PROGRAM PRG_CohapTest
VAR
END_VAR

ACTION A_InitCohapMethodParams:
strDeviceName := 'Device12133';

readSerialNumber_inpuparams[0].strKey := 'channel';
readSerialNumber_inpuparams[0].strValue := '1';
readSerialNumber_inpuparams[1].strKey := '';
readSerialNumber_inpuparams[1].strValue := '';
readSerialNumber_inpuparams[2].strKey := '';
readSerialNumber_inpuparams[2].strValue := '';

readSerialNumber_expoutparamlist[0].enumDataType := E_DataType.DT_ULINT;
readSerialNumber_expoutparamlist[0].strVarName := 'serialnumber';
readSerialNumber_expoutparamlist[1].enumDataType := E_DataType.DT_STRING;
readSerialNumber_expoutparamlist[1].strVarName := 'stringserialno';
readSerialNumber_expoutparamlist[2].enumDataType := E_DataType.DT_STRING;
readSerialNumber_expoutparamlist[2].strVarName := '';


ReadDeviceOutput_inpuparams[0].strKey := 'channel';
ReadDeviceOutput_inpuparams[0].strValue := '1';
ReadDeviceOutput_inpuparams[1].strKey := '';
ReadDeviceOutput_inpuparams[1].strValue := '';
ReadDeviceOutput_inpuparams[2].strKey := '';
ReadDeviceOutput_inpuparams[2].strValue := '';

ReadDeviceOutput_expoutparamlist[0].enumDataType := E_DataType.DT_INT;
ReadDeviceOutput_expoutparamlist[0].strVarName := 'P1data';
ReadDeviceOutput_expoutparamlist[1].enumDataType := E_DataType.DT_INT;
ReadDeviceOutput_expoutparamlist[1].strVarName := 'P1out';
ReadDeviceOutput_expoutparamlist[2].enumDataType := E_DataType.DT_INT;
ReadDeviceOutput_expoutparamlist[2].strVarName := 'P2data';
ReadDeviceOutput_expoutparamlist[3].enumDataType := E_DataType.DT_INT;
ReadDeviceOutput_expoutparamlist[3].strVarName := 'P2out';
ReadDeviceOutput_expoutparamlist[4].enumDataType := E_DataType.DT_INT;
ReadDeviceOutput_expoutparamlist[4].strVarName := 'T1data';
ReadDeviceOutput_expoutparamlist[5].enumDataType := E_DataType.DT_INT;
ReadDeviceOutput_expoutparamlist[5].strVarName := 'T1out';
ReadDeviceOutput_expoutparamlist[6].enumDataType := E_DataType.DT_INT;
ReadDeviceOutput_expoutparamlist[6].strVarName := 'T2data';
ReadDeviceOutput_expoutparamlist[7].enumDataType := E_DataType.DT_INT;
ReadDeviceOutput_expoutparamlist[7].strVarName := 'T2out';

PowerUp_inpuparams[0].strKey := 'channel';
PowerUp_inpuparams[0].strValue := '1';
PowerUp_inpuparams[1].strKey := 'supplyVoltage';
PowerUp_inpuparams[1].strValue := '5.0';
PowerUp_inpuparams[2].strKey := '';
PowerUp_inpuparams[2].strValue := '';

PowerUp_expoutparamlist[0].enumDataType := E_DataType.DT_DOUBLE;
PowerUp_expoutparamlist[0].strVarName := 'Vsupply';
PowerUp_expoutparamlist[1].enumDataType := E_DataType.DT_DOUBLE;
PowerUp_expoutparamlist[1].strVarName := 'current';
PowerUp_expoutparamlist[2].enumDataType := E_DataType.DT_STRING;
PowerUp_expoutparamlist[2].strVarName := '';

PowerDown_inpuparams[0].strKey := 'channel';
PowerDown_inpuparams[0].strValue := '1';
PowerDown_inpuparams[1].strKey := '';
PowerDown_inpuparams[1].strValue := '';
PowerDown_inpuparams[2].strKey := '';
PowerDown_inpuparams[2].strValue := '';

PowerDown_expoutparamlist[0].enumDataType := E_DataType.DT_STRING;
PowerDown_expoutparamlist[0].strVarName := '';
PowerDown_expoutparamlist[1].enumDataType := E_DataType.DT_STRING;
PowerDown_expoutparamlist[1].strVarName := '';
PowerDown_expoutparamlist[2].enumDataType := E_DataType.DT_STRING;
PowerDown_expoutparamlist[2].strVarName := '';

TestDummy_inpuparams[0].strKey := 'channel';
TestDummy_inpuparams[0].strValue := '1';
TestDummy_inpuparams[1].strKey := 'bInput';
TestDummy_inpuparams[1].strValue := 'FALSE';
TestDummy_inpuparams[2].strKey := '';
TestDummy_inpuparams[2].strValue := '';

TestDummy_expoutparamlist[0].enumDataType := E_DataType.DT_STRING;
TestDummy_expoutparamlist[0].strVarName := 'serialno';
TestDummy_expoutparamlist[1].enumDataType := E_DataType.DT_DOUBLE;
TestDummy_expoutparamlist[1].strVarName := 'Voltage';
TestDummy_expoutparamlist[2].enumDataType := E_DataType.DT_BOOL;
TestDummy_expoutparamlist[2].strVarName := 'MethodResponse';
TestDummy_expoutparamlist[3].enumDataType := E_DataType.DT_UINT;
TestDummy_expoutparamlist[3].strVarName := 'current';
TestDummy_expoutparamlist[4].enumDataType := E_DataType.DT_STRING;
TestDummy_expoutparamlist[4].strVarName := 'P1status';
TestDummy_expoutparamlist[5].enumDataType := E_DataType.DT_STRING;
TestDummy_expoutparamlist[5].strVarName := 'P2status';

TestDummy2_inpuparams[0].strKey := 'channel';
TestDummy2_inpuparams[0].strValue := '1';
TestDummy2_inpuparams[1].strKey := 'Input2';
TestDummy2_inpuparams[1].strValue := 'dummyimput2';
TestDummy2_inpuparams[2].strKey := '';
TestDummy2_inpuparams[2].strValue := '';

TestDummy2_expoutparamlist[0].enumDataType := E_DataType.DT_INT;
TestDummy2_expoutparamlist[0].strVarName := 'output1';
TestDummy2_expoutparamlist[1].enumDataType := E_DataType.DT_STRING;
TestDummy2_expoutparamlist[1].strVarName := 'output2';
TestDummy2_expoutparamlist[2].enumDataType := E_DataType.DT_ULINT;
TestDummy2_expoutparamlist[2].strVarName := 'fastchannel1';
TestDummy2_expoutparamlist[3].enumDataType := E_DataType.DT_ULINT;
TestDummy2_expoutparamlist[3].strVarName := 'fastchannel2';
TestDummy2_expoutparamlist[4].enumDataType := E_DataType.DT_STRING;
TestDummy2_expoutparamlist[4].strVarName := 'fastchannel3';
TestDummy2_expoutparamlist[5].enumDataType := E_DataType.DT_INT;
TestDummy2_expoutparamlist[5].strVarName := 'fastchannel4';
TestDummy2_expoutparamlist[6].enumDataType := E_DataType.DT_ULINT;
TestDummy2_expoutparamlist[6].strVarName := 'fastchannel5';
TestDummy2_expoutparamlist[7].enumDataType := E_DataType.DT_ULINT;
TestDummy2_expoutparamlist[7].strVarName := 'fastchannel6';
TestDummy2_expoutparamlist[8].enumDataType := E_DataType.DT_STRING;
TestDummy2_expoutparamlist[8].strVarName := 'fastchannel7';
TestDummy2_expoutparamlist[9].enumDataType := E_DataType.DT_INT;
TestDummy2_expoutparamlist[9].strVarName := 'fastchannel8';

//TestDummy2_outputparams[0].strKey := '';
//TestDummy2_outputparams[0].strValue := '';
//TestDummy2_outputparams[1].strKey := '';
//TestDummy2_outputparams[1].strValue := '';
//TestDummy2_outputparams[2].strKey := '';
//TestDummy2_outputparams[2].strValue := '';
//TestDummy2_outputparams[3].strKey := '';
//TestDummy2_outputparams[3].strValue := '';
//TestDummy2_outputparams[4].strKey := '';
//TestDummy2_outputparams[4].strValue := '';
//TestDummy2_outputparams[5].strKey := '';
//TestDummy2_outputparams[5].strValue := '';
//TestDummy2_outputparams[6].strKey := '';
//TestDummy2_outputparams[6].strValue := '';
//TestDummy2_outputparams[7].strKey := '';
//TestDummy2_outputparams[7].strValue := '';
//TestDummy2_outputparams[8].strKey := '';
//TestDummy2_outputparams[8].strValue := '';
//TestDummy2_outputparams[9].strKey := '';
//TestDummy2_outputparams[9].strValue := '';

init_inpuparams[0].strKey := 'VSupply';
init_inpuparams[0].strValue := '5.0';
init_inpuparams[1].strKey := '';
init_inpuparams[1].strValue := '';
init_inpuparams[2].strKey := '';
init_inpuparams[2].strValue := '';

init_expoutparamlist[0].enumDataType := E_DataType.DT_STRING;
init_expoutparamlist[0].strVarName := 'returnMsg';
init_expoutparamlist[1].enumDataType := E_DataType.DT_STRING;
init_expoutparamlist[1].strVarName := '';
init_expoutparamlist[2].enumDataType := E_DataType.DT_STRING;
init_expoutparamlist[2].strVarName := '';

getSICAndChannelCardVersions_inpuparams[0].strKey := 'channel';
getSICAndChannelCardVersions_inpuparams[0].strValue := '1';
getSICAndChannelCardVersions_inpuparams[1].strKey := '';
getSICAndChannelCardVersions_inpuparams[1].strValue := '';
getSICAndChannelCardVersions_inpuparams[2].strKey := '';
getSICAndChannelCardVersions_inpuparams[2].strValue := '';

getSICAndChannelCardVersions_expoutparamlist[0].enumDataType := E_DataType.DT_STRING;
getSICAndChannelCardVersions_expoutparamlist[0].strVarName := 'SICVersion';
getSICAndChannelCardVersions_expoutparamlist[1].enumDataType := E_DataType.DT_STRING;
getSICAndChannelCardVersions_expoutparamlist[1].strVarName := 'COHAPChannelCardVersion';
getSICAndChannelCardVersions_expoutparamlist[2].enumDataType := E_DataType.DT_STRING;
getSICAndChannelCardVersions_expoutparamlist[2].strVarName := '';

getDLLVersions_inpuparams[0].strKey := '';
getDLLVersions_inpuparams[0].strValue := '';
getDLLVersions_inpuparams[1].strKey := '';
getDLLVersions_inpuparams[1].strValue := '';
getDLLVersions_inpuparams[2].strKey := '';
getDLLVersions_inpuparams[2].strValue := '';

getDLLVersions_expoutparamlist[0].enumDataType := E_DataType.DT_STRING;
getDLLVersions_expoutparamlist[0].strVarName := 'DUT12133DLLVersion';
getDLLVersions_expoutparamlist[1].enumDataType := E_DataType.DT_STRING;
getDLLVersions_expoutparamlist[1].strVarName := 'MUPeT12133DLLVersion';
getDLLVersions_expoutparamlist[2].enumDataType := E_DataType.DT_STRING;
getDLLVersions_expoutparamlist[2].strVarName := 'HALDLLVersion';


initDUT_inpuparams[0].strKey := 'channel';
initDUT_inpuparams[0].strValue := '1';
initDUT_inpuparams[1].strKey := 'supplyVoltage';
initDUT_inpuparams[1].strValue := '5.0';
initDUT_inpuparams[2].strKey := '';
initDUT_inpuparams[2].strValue := '';

initDUT_expoutparamlist[0].enumDataType := E_DataType.DT_STRING;
initDUT_expoutparamlist[0].strVarName := '';
initDUT_expoutparamlist[1].enumDataType := E_DataType.DT_STRING;
initDUT_expoutparamlist[1].strVarName := '';
initDUT_expoutparamlist[2].enumDataType := E_DataType.DT_STRING;
initDUT_expoutparamlist[2].strVarName := '';


readFastChannelData_inputparams[0].strKey := 'channel';
readFastChannelData_inputparams[0].strValue := '1';
readFastChannelData_inputparams[1].strKey := '';
readFastChannelData_inputparams[1].strValue := '';
readFastChannelData_inputparams[2].strKey := '';
readFastChannelData_inputparams[2].strValue := '';

readFastChannelData_expoutparamlist[0].enumDataType := E_DataType.DT_UINT;
readFastChannelData_expoutparamlist[0].strVarName := 'FastChannel1Data';
readFastChannelData_expoutparamlist[1].enumDataType := E_DataType.DT_UINT;
readFastChannelData_expoutparamlist[1].strVarName := 'FastChannel2Data';
readFastChannelData_expoutparamlist[2].enumDataType := E_DataType.DT_STRING;
readFastChannelData_expoutparamlist[2].strVarName := 'FastChannel1Status';
readFastChannelData_expoutparamlist[3].enumDataType := E_DataType.DT_STRING;
readFastChannelData_expoutparamlist[3].strVarName := 'FastChannel2Status';


InitLot_inputparams[0].strKey := 'deviceID';
InitLot_inputparams[0].strValue := '52EMB01-01';
InitLot_inputparams[1].strKey := 'lotID';
InitLot_inputparams[1].strValue := '123';
InitLot_inputparams[2].strKey := 'equipmentID';
InitLot_inputparams[2].strValue := '1';
InitLot_inputparams[3].strKey := 'testKind';
InitLot_inputparams[3].strValue := '1';

t1Precal_inputparams[0].strKey := 'channel';
t1Precal_inputparams[0].strValue := '1';
t1Precal_inputparams[1].strKey := 'deviceID';
t1Precal_inputparams[1].strValue := '52EMB01-01';
t1Precal_inputparams[2].strKey := 'temperature';
t1Precal_inputparams[2].strValue := '-25';
t1Precal_inputparams[3].strKey := 'force';
t1Precal_inputparams[3].strValue := '0';
 
t1Step2_inputparams[0].strKey := 'deviceID';
t1Step2_inputparams[0].strValue := '52EMB01-01';
t1Step2_inputparams[1].strKey := 'temperature';
t1Step2_inputparams[1].strValue := '-25';
t1Step2_inputparams[2].strKey := 'force';
t1Step2_inputparams[2].strValue := '40';
 
t1Step3_inputparams[0].strKey := 'deviceID';
t1Step3_inputparams[0].strValue := '52EMB01-01';
t1Step3_inputparams[2].strKey := 'temperature';
t1Step3_inputparams[2].strValue := '-25';
t1Step3_inputparams[3].strKey := 'force';
t1Step3_inputparams[3].strValue := '0';
END_ACTION

METHOD M_TestCohapLibrary : BOOL
VAR_INPUT
END_VAR
VAR
	//Testing Cohap Related Vars

	//Initialize Only	
	MyCohapTest : FB_COHAP;
	bInitializeCohapSystem: BOOL;
	bRes_CohapConnected: BOOL;

	//Execute RunImpMethods Only	;
	bExecuteRunImpMethods: BOOL;
	bRes_RunImpMethods: BOOL;

	//Set Current Device Instance
	bSetCurrentDevice_Cohap : BOOL;
	bRes_SetCurrentDevice : BOOL;
	//Input Params
	strDeviceName : STRING;
	
	//RunCommand
	bRunCommandCohapSystem : BOOL;
	bRes_RunCommand : BOOL;
	//Input Params
	strMethodName : STRING;
	RunCom_InpuParams : T_CohapParameterList;
	RunCom_ExpOutParamList : ARRAY[0..9] OF ST_ReturnParamsInfo;
	//Output Params
	RunCom_OutputParams : T_CohapParameterList;
	
	//DummyTest Dictionary Prep for RunCommand Execution
	RC_DT_InpPar : T_CohapParameterList;
	RC_DT_ExpOutPL : ARRAY[0..9] OF ST_ReturnParamsInfo;
	
	CohapMethodStrings : TMethodNames_Cohap;
	CohapMethodControls : TMethod_Controls;
//	fbCohapHandler1: FB_COHAP;

///////////////////////////////

	// For readSerialNumber
	readSerialNumber_inpuparams : T_CohapParameterList;
	readSerialNumber_expoutparamlist : ARRAY[0..9] OF ST_ReturnParamsInfo;
	readSerialNumber_outputparams : T_CohapParameterList;
	
	// For ReadDeviceOutput
	ReadDeviceOutput_inpuparams : T_CohapParameterList;
	ReadDeviceOutput_expoutparamlist : ARRAY[0..9] OF ST_ReturnParamsInfo;
	ReadDeviceOutput_outputparams : T_CohapParameterList;

	
	// For PowerUp
	PowerUp_inpuparams : T_CohapParameterList;
	PowerUp_expoutparamlist : ARRAY[0..9] OF ST_ReturnParamsInfo;
	PowerUp_outputparams : T_CohapParameterList;
	
	// For PowerDown
	PowerDown_inpuparams : T_CohapParameterList;
	PowerDown_expoutparamlist : ARRAY[0..9] OF ST_ReturnParamsInfo;
	PowerDown_outputparams : T_CohapParameterList;
	
	// For TestDummy
	TestDummy_inpuparams : T_CohapParameterList;
	TestDummy_expoutparamlist : ARRAY[0..9] OF ST_ReturnParamsInfo;
	TestDummy_outputparams : T_CohapParameterList;
	
	// For TestDummy2
	TestDummy2_inpuparams : T_CohapParameterList;
	TestDummy2_expoutparamlist : ARRAY[0..9] OF ST_ReturnParamsInfo;
	TestDummy2_outputparams : T_CohapParameterList;
	
	// For init
	init_inpuparams : T_CohapParameterList;
	init_expoutparamlist : ARRAY[0..9] OF ST_ReturnParamsInfo;
	init_outputparams : T_CohapParameterList;
	
	// For getSICAndChannelCardVersions
	getSICAndChannelCardVersions_inpuparams : T_CohapParameterList;
	getSICAndChannelCardVersions_expoutparamlist : ARRAY[0..9] OF ST_ReturnParamsInfo;
	getSICAndChannelCardVersions_outputparams : T_CohapParameterList;
	
	// For getDLLVersions
	getDLLVersions_inpuparams : T_CohapParameterList;
	getDLLVersions_expoutparamlist : ARRAY[0..9] OF ST_ReturnParamsInfo;
	getDLLVersions_outputparams : T_CohapParameterList;
	
	// For initDUT
	initDUT_inpuparams : T_CohapParameterList;
	initDUT_expoutparamlist : ARRAY[0..9] OF ST_ReturnParamsInfo;
	initDUT_outputparams : T_CohapParameterList;
	
	//For Fast Channel Data
	readFastChannelData_inputparams : T_CohapParameterList;
	readFastChannelData_expoutparamlist : ARRAY[0..9] OF ST_ReturnParamsInfo;
	readFastChannelData_outputparams : T_CohapParameterList;

	// For T1 Step 1 Calibration
	t1Step1_inpuparams : T_CohapParameterList;
	t1Step1_expoutparamlist : ARRAY[0..9] OF ST_ReturnParamsInfo;
	t1Step1_outputparams : T_CohapParameterList;
	
//	// For T1 Step 2 Calibration
//	t1Step2_inpuparams : T_CohapParameterList;
//	t1Step2_expoutparamlist : ARRAY[0..9] OF ST_ReturnParamsInfo;
//	t1Step2_outputparams : T_CohapParameterList;
	
//	// For T1 Step 3 Calibration
//	t1Step3_inpuparams : T_CohapParameterList;
//	t1Step3_expoutparamlist : ARRAY[0..9] OF ST_ReturnParamsInfo;
//	t1Step3_outputparams : T_CohapParameterList;
	
	// For T2 Step 1 Calibration
	t2Step1_inpuparams : T_CohapParameterList;
	t2Step1_expoutparamlist : ARRAY[0..9] OF ST_ReturnParamsInfo;
	t2Step1_outputparams : T_CohapParameterList;
	
	// For T2 Step 2 Calibration
	t2Step2_inpuparams : T_CohapParameterList;
	t2Step2_expoutparamlist : ARRAY[0..9] OF ST_ReturnParamsInfo;
	t2Step2_outputparams : T_CohapParameterList;
	
	// For T2 Step 3 Calibration
	t2Step3_inpuparams : T_CohapParameterList;
	t2Step3_expoutparamlist : ARRAY[0..9] OF ST_ReturnParamsInfo;
	t2Step3_outputparams : T_CohapParameterList;
	
	// InitLot Device12133 class in Mech Device Lib Calibration
	InitLot_inputparams : T_CohapParameterList;
	InitLot_expoutparamlist : ARRAY[0..9] OF ST_ReturnParamsInfo;
	InitLot_outputparams : T_CohapParameterList;
	
//	//For Init Lot
//	InitLot_inputparams : T_CohapParameterList;
//	InitLot_expoutparamlist : ARRAY[0..9] OF ST_ReturnParamsInfo;
//	InitLot_outputparams : T_CohapParameterList;	
	// For T1 Step 1 Calibration
	t1Precal_inputparams : T_CohapParameterList;
	t1Precal_expoutparamlist : ARRAY[0..9] OF ST_ReturnParamsInfo;
	t1Precal_outputparams : T_CohapParameterList;
	// For T1 Step 2 Calibration
	t1Step2_inputparams : T_CohapParameterList;
	t1Step2_expoutparamlist : ARRAY[0..9] OF ST_ReturnParamsInfo;
	t1Step2_outputparams : T_CohapParameterList;
	// For T1 Step 3 Calibration
	t1Step3_inputparams : T_CohapParameterList;
	t1Step3_expoutparamlist : ARRAY[0..9] OF ST_ReturnParamsInfo;
	t1Step3_outputparams : T_CohapParameterList;
END_VAR
VAR_INST // added by the converter: edge detectors and wires of the graphical bodies
    _w1, _w2, _w3, _w4, _w5, _w6, _w7, _w8, _w9, _w10, _w11, _w12, _w13, _w14, _w15, _w16, _w17, _w18, _w19, _w20, _w21, _w22, _w23, _w24, _w25, _w26, _w27, _w28, _w29, _w30, _w31, _w32, _w33, _w34, _w35, _w36, _w37, _w38, _w39, _w40 : BOOL;
END_VAR
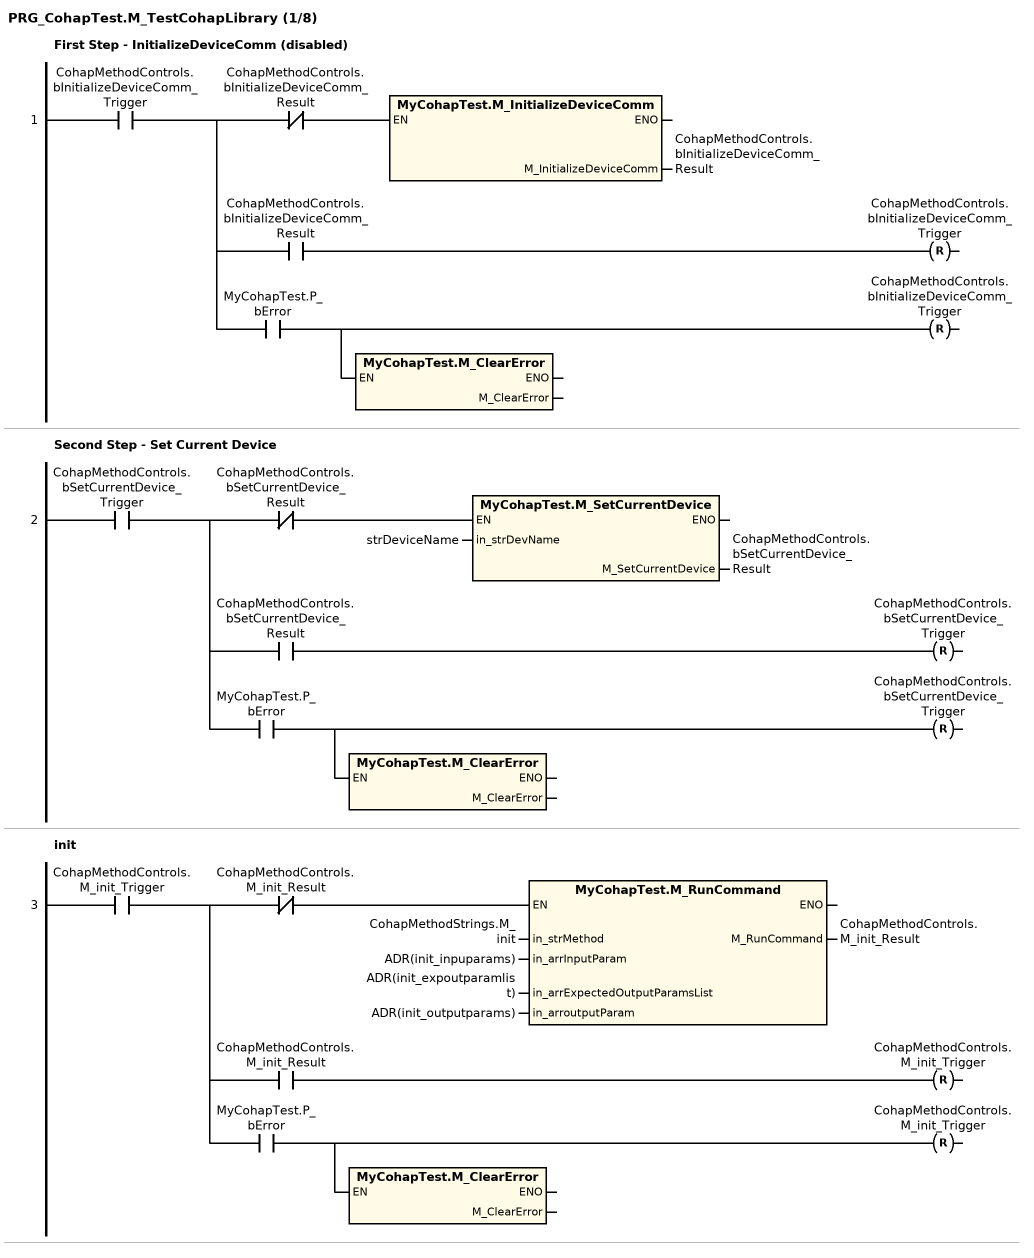
// NETWORK 1: First Step - InitializeDeviceComm (disabled)
// _w1 := CohapMethodControls.bInitializeDeviceComm_Trigger;
// IF _w1 AND NOT CohapMethodControls.bInitializeDeviceComm_Result THEN
//     CohapMethodControls.bInitializeDeviceComm_Result := MyCohapTest.M_InitializeDeviceComm();
// END_IF
// CohapMethodControls.bInitializeDeviceComm_Trigger R= _w1 AND CohapMethodControls.bInitializeDeviceComm_Result;
// _w2 := _w1 AND MyCohapTest.P_bError;
// CohapMethodControls.bInitializeDeviceComm_Trigger R= _w2;
// IF _w2 THEN MyCohapTest.M_ClearError(); END_IF

// NETWORK 2: Second Step - Set Current Device
_w3 := CohapMethodControls.bSetCurrentDevice_Trigger;
IF _w3 AND NOT CohapMethodControls.bSetCurrentDevice_Result THEN
    CohapMethodControls.bSetCurrentDevice_Result := MyCohapTest.M_SetCurrentDevice(in_strDevName := strDeviceName);
END_IF
CohapMethodControls.bSetCurrentDevice_Trigger R= _w3 AND CohapMethodControls.bSetCurrentDevice_Result;
_w4 := _w3 AND MyCohapTest.P_bError;
CohapMethodControls.bSetCurrentDevice_Trigger R= _w4;
IF _w4 THEN MyCohapTest.M_ClearError(); END_IF

// NETWORK 3: init
_w5 := CohapMethodControls.M_init_Trigger;
IF _w5 AND NOT CohapMethodControls.M_init_Result THEN
    CohapMethodControls.M_init_Result := MyCohapTest.M_RunCommand(in_strMethod := CohapMethodStrings.M_init, in_arrInputParam := ADR(init_inpuparams), in_arrExpectedOutputParamsList := ADR(init_expoutparamlist), in_arroutputParam := ADR(init_outputparams));
END_IF
CohapMethodControls.M_init_Trigger R= _w5 AND CohapMethodControls.M_init_Result;
_w6 := _w5 AND MyCohapTest.P_bError;
CohapMethodControls.M_init_Trigger R= _w6;
IF _w6 THEN MyCohapTest.M_ClearError(); END_IF

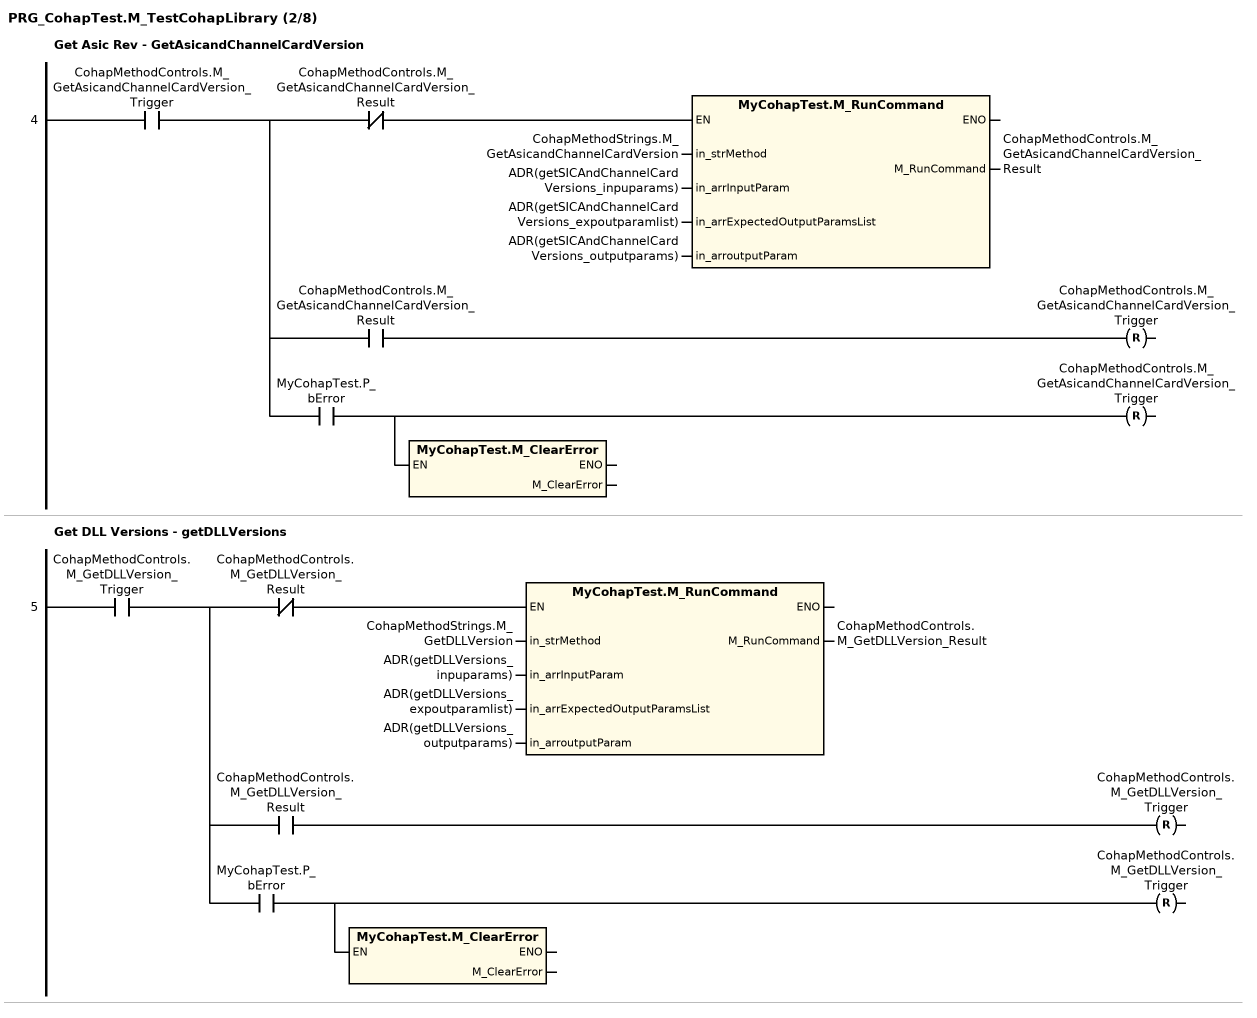
// NETWORK 4: Get Asic Rev - GetAsicandChannelCardVersion
_w7 := CohapMethodControls.M_GetAsicandChannelCardVersion_Trigger;
IF _w7 AND NOT CohapMethodControls.M_GetAsicandChannelCardVersion_Result THEN
    CohapMethodControls.M_GetAsicandChannelCardVersion_Result := MyCohapTest.M_RunCommand(in_strMethod := CohapMethodStrings.M_GetAsicandChannelCardVersion, in_arrInputParam := ADR(getSICAndChannelCardVersions_inpuparams), in_arrExpectedOutputParamsList := ADR(getSICAndChannelCardVersions_expoutparamlist), in_arroutputParam := ADR(getSICAndChannelCardVersions_outputparams));
END_IF
CohapMethodControls.M_GetAsicandChannelCardVersion_Trigger R= _w7 AND CohapMethodControls.M_GetAsicandChannelCardVersion_Result;
_w8 := _w7 AND MyCohapTest.P_bError;
CohapMethodControls.M_GetAsicandChannelCardVersion_Trigger R= _w8;
IF _w8 THEN MyCohapTest.M_ClearError(); END_IF

// NETWORK 5: Get DLL Versions - getDLLVersions
_w9 := CohapMethodControls.M_GetDLLVersion_Trigger;
IF _w9 AND NOT CohapMethodControls.M_GetDLLVersion_Result THEN
    CohapMethodControls.M_GetDLLVersion_Result := MyCohapTest.M_RunCommand(in_strMethod := CohapMethodStrings.M_GetDLLVersion, in_arrInputParam := ADR(getDLLVersions_inpuparams), in_arrExpectedOutputParamsList := ADR(getDLLVersions_expoutparamlist), in_arroutputParam := ADR(getDLLVersions_outputparams));
END_IF
CohapMethodControls.M_GetDLLVersion_Trigger R= _w9 AND CohapMethodControls.M_GetDLLVersion_Result;
_w10 := _w9 AND MyCohapTest.P_bError;
CohapMethodControls.M_GetDLLVersion_Trigger R= _w10;
IF _w10 THEN MyCohapTest.M_ClearError(); END_IF

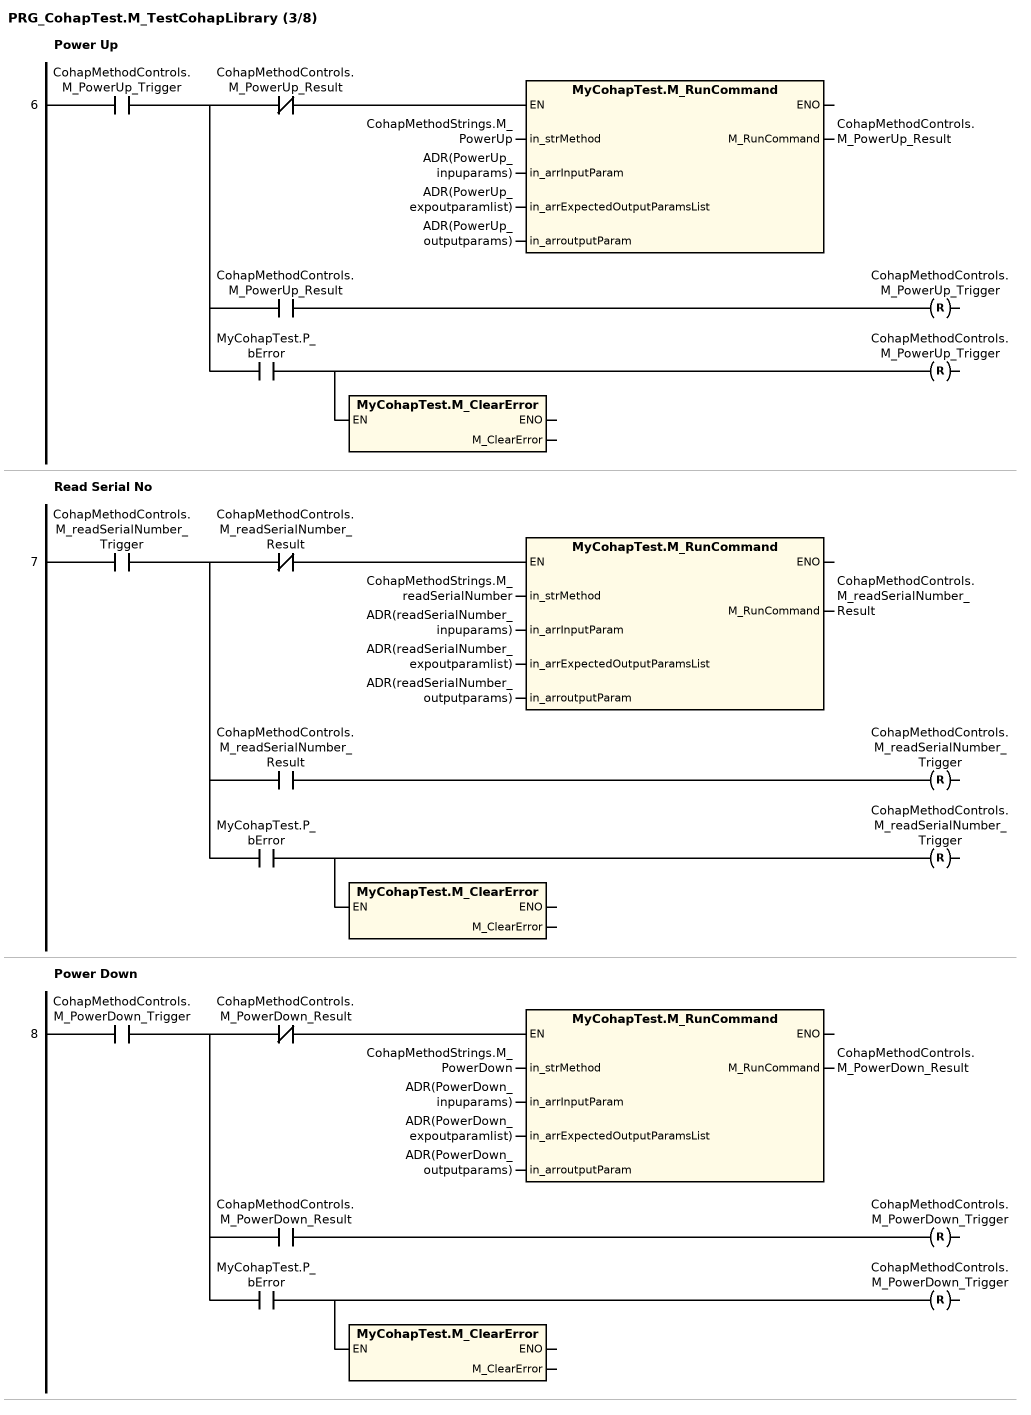
// NETWORK 6: Power Up
_w11 := CohapMethodControls.M_PowerUp_Trigger;
IF _w11 AND NOT CohapMethodControls.M_PowerUp_Result THEN
    CohapMethodControls.M_PowerUp_Result := MyCohapTest.M_RunCommand(in_strMethod := CohapMethodStrings.M_PowerUp, in_arrInputParam := ADR(PowerUp_inpuparams), in_arrExpectedOutputParamsList := ADR(PowerUp_expoutparamlist), in_arroutputParam := ADR(PowerUp_outputparams));
END_IF
CohapMethodControls.M_PowerUp_Trigger R= _w11 AND CohapMethodControls.M_PowerUp_Result;
_w12 := _w11 AND MyCohapTest.P_bError;
CohapMethodControls.M_PowerUp_Trigger R= _w12;
IF _w12 THEN MyCohapTest.M_ClearError(); END_IF

// NETWORK 7: Read Serial No
_w13 := CohapMethodControls.M_readSerialNumber_Trigger;
IF _w13 AND NOT CohapMethodControls.M_readSerialNumber_Result THEN
    CohapMethodControls.M_readSerialNumber_Result := MyCohapTest.M_RunCommand(in_strMethod := CohapMethodStrings.M_readSerialNumber, in_arrInputParam := ADR(readSerialNumber_inpuparams), in_arrExpectedOutputParamsList := ADR(readSerialNumber_expoutparamlist), in_arroutputParam := ADR(readSerialNumber_outputparams));
END_IF
CohapMethodControls.M_readSerialNumber_Trigger R= _w13 AND CohapMethodControls.M_readSerialNumber_Result;
_w14 := _w13 AND MyCohapTest.P_bError;
CohapMethodControls.M_readSerialNumber_Trigger R= _w14;
IF _w14 THEN MyCohapTest.M_ClearError(); END_IF

// NETWORK 8: Power Down
_w15 := CohapMethodControls.M_PowerDown_Trigger;
IF _w15 AND NOT CohapMethodControls.M_PowerDown_Result THEN
    CohapMethodControls.M_PowerDown_Result := MyCohapTest.M_RunCommand(in_strMethod := CohapMethodStrings.M_PowerDown, in_arrInputParam := ADR(PowerDown_inpuparams), in_arrExpectedOutputParamsList := ADR(PowerDown_expoutparamlist), in_arroutputParam := ADR(PowerDown_outputparams));
END_IF
CohapMethodControls.M_PowerDown_Trigger R= _w15 AND CohapMethodControls.M_PowerDown_Result;
_w16 := _w15 AND MyCohapTest.P_bError;
CohapMethodControls.M_PowerDown_Trigger R= _w16;
IF _w16 THEN MyCohapTest.M_ClearError(); END_IF

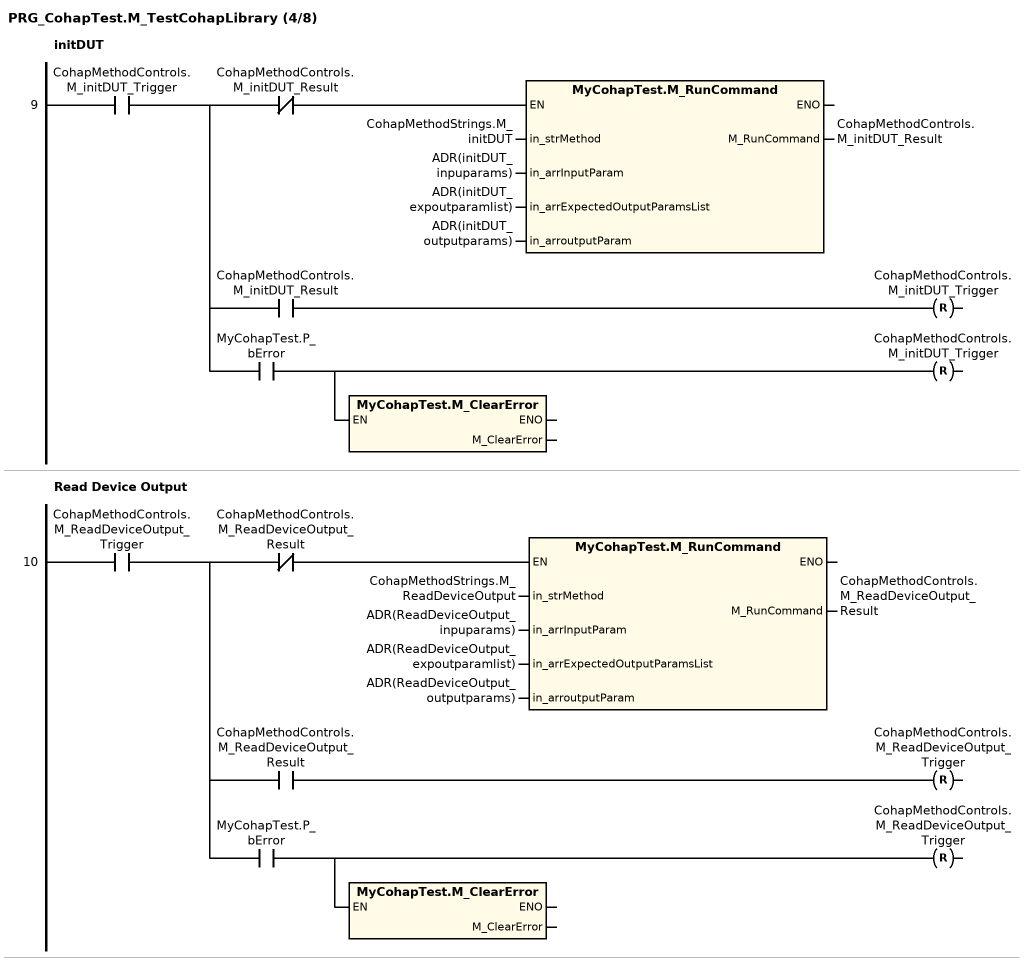
// NETWORK 9: initDUT
_w17 := CohapMethodControls.M_initDUT_Trigger;
IF _w17 AND NOT CohapMethodControls.M_initDUT_Result THEN
    CohapMethodControls.M_initDUT_Result := MyCohapTest.M_RunCommand(in_strMethod := CohapMethodStrings.M_initDUT, in_arrInputParam := ADR(initDUT_inpuparams), in_arrExpectedOutputParamsList := ADR(initDUT_expoutparamlist), in_arroutputParam := ADR(initDUT_outputparams));
END_IF
CohapMethodControls.M_initDUT_Trigger R= _w17 AND CohapMethodControls.M_initDUT_Result;
_w18 := _w17 AND MyCohapTest.P_bError;
CohapMethodControls.M_initDUT_Trigger R= _w18;
IF _w18 THEN MyCohapTest.M_ClearError(); END_IF

// NETWORK 10: Read Device Output
_w19 := CohapMethodControls.M_ReadDeviceOutput_Trigger;
IF _w19 AND NOT CohapMethodControls.M_ReadDeviceOutput_Result THEN
    CohapMethodControls.M_ReadDeviceOutput_Result := MyCohapTest.M_RunCommand(in_strMethod := CohapMethodStrings.M_ReadDeviceOutput, in_arrInputParam := ADR(ReadDeviceOutput_inpuparams), in_arrExpectedOutputParamsList := ADR(ReadDeviceOutput_expoutparamlist), in_arroutputParam := ADR(ReadDeviceOutput_outputparams));
END_IF
CohapMethodControls.M_ReadDeviceOutput_Trigger R= _w19 AND CohapMethodControls.M_ReadDeviceOutput_Result;
_w20 := _w19 AND MyCohapTest.P_bError;
CohapMethodControls.M_ReadDeviceOutput_Trigger R= _w20;
IF _w20 THEN MyCohapTest.M_ClearError(); END_IF

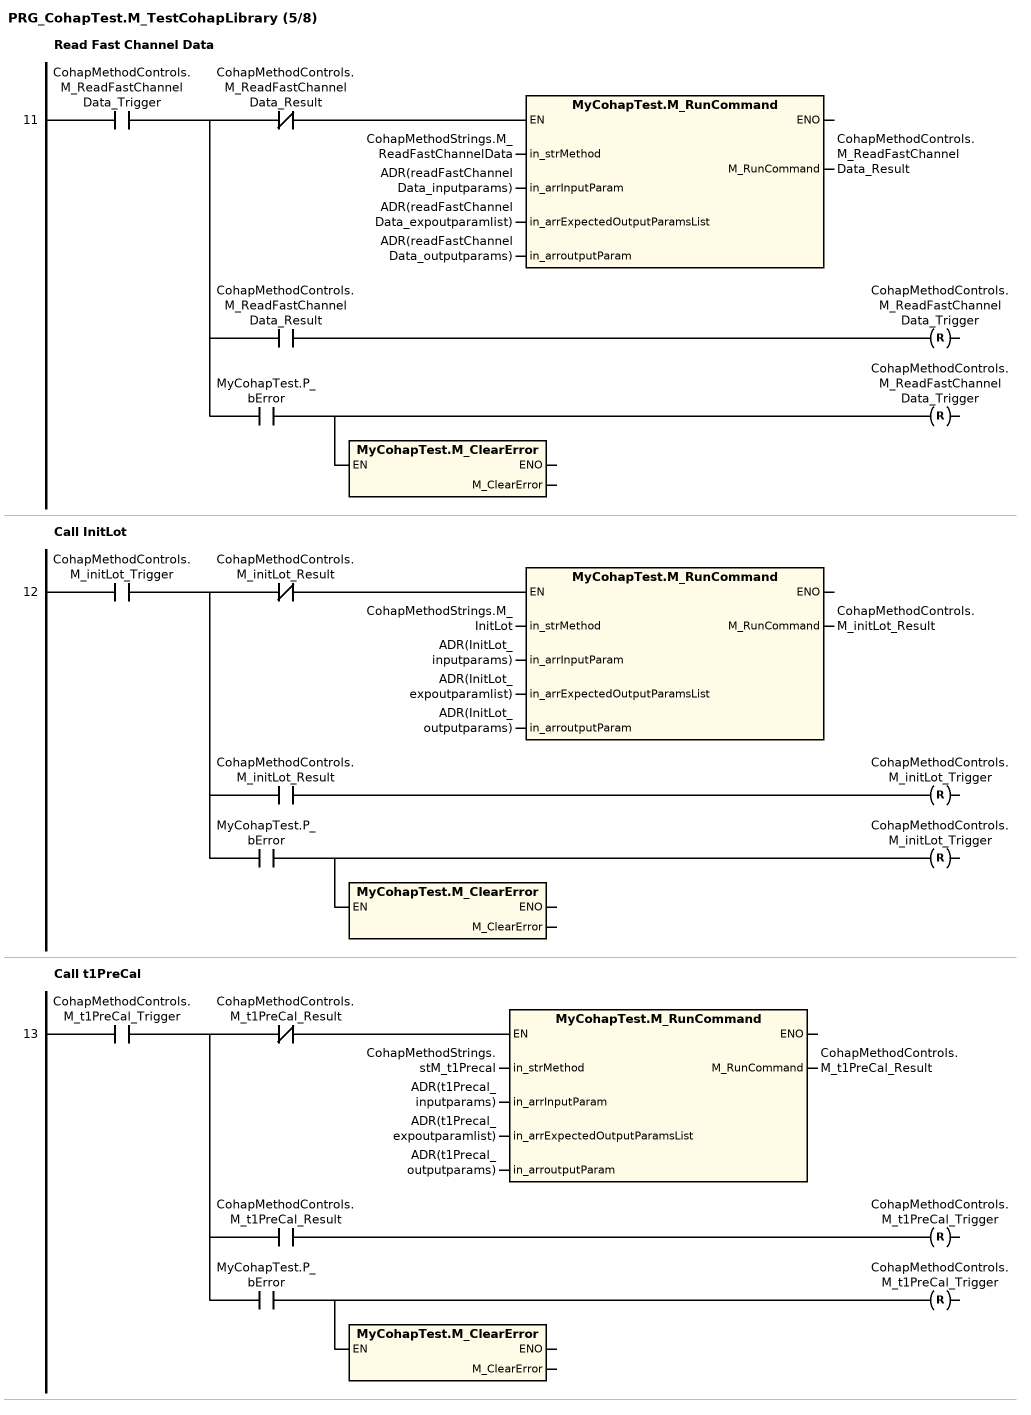
// NETWORK 11: Read Fast Channel Data
_w21 := CohapMethodControls.M_ReadFastChannelData_Trigger;
IF _w21 AND NOT CohapMethodControls.M_ReadFastChannelData_Result THEN
    CohapMethodControls.M_ReadFastChannelData_Result := MyCohapTest.M_RunCommand(in_strMethod := CohapMethodStrings.M_ReadFastChannelData, in_arrInputParam := ADR(readFastChannelData_inputparams), in_arrExpectedOutputParamsList := ADR(readFastChannelData_expoutparamlist), in_arroutputParam := ADR(readFastChannelData_outputparams));
END_IF
CohapMethodControls.M_ReadFastChannelData_Trigger R= _w21 AND CohapMethodControls.M_ReadFastChannelData_Result;
_w22 := _w21 AND MyCohapTest.P_bError;
CohapMethodControls.M_ReadFastChannelData_Trigger R= _w22;
IF _w22 THEN MyCohapTest.M_ClearError(); END_IF

// NETWORK 12: Call InitLot
_w23 := CohapMethodControls.M_initLot_Trigger;
IF _w23 AND NOT CohapMethodControls.M_initLot_Result THEN
    CohapMethodControls.M_initLot_Result := MyCohapTest.M_RunCommand(in_strMethod := CohapMethodStrings.M_InitLot, in_arrInputParam := ADR(InitLot_inputparams), in_arrExpectedOutputParamsList := ADR(InitLot_expoutparamlist), in_arroutputParam := ADR(InitLot_outputparams));
END_IF
CohapMethodControls.M_initLot_Trigger R= _w23 AND CohapMethodControls.M_initLot_Result;
_w24 := _w23 AND MyCohapTest.P_bError;
CohapMethodControls.M_initLot_Trigger R= _w24;
IF _w24 THEN MyCohapTest.M_ClearError(); END_IF

// NETWORK 13: Call t1PreCal
_w25 := CohapMethodControls.M_t1PreCal_Trigger;
IF _w25 AND NOT CohapMethodControls.M_t1PreCal_Result THEN
    CohapMethodControls.M_t1PreCal_Result := MyCohapTest.M_RunCommand(in_strMethod := CohapMethodStrings.stM_t1Precal, in_arrInputParam := ADR(t1Precal_inputparams), in_arrExpectedOutputParamsList := ADR(t1Precal_expoutparamlist), in_arroutputParam := ADR(t1Precal_outputparams));
END_IF
CohapMethodControls.M_t1PreCal_Trigger R= _w25 AND CohapMethodControls.M_t1PreCal_Result;
_w26 := _w25 AND MyCohapTest.P_bError;
CohapMethodControls.M_t1PreCal_Trigger R= _w26;
IF _w26 THEN MyCohapTest.M_ClearError(); END_IF

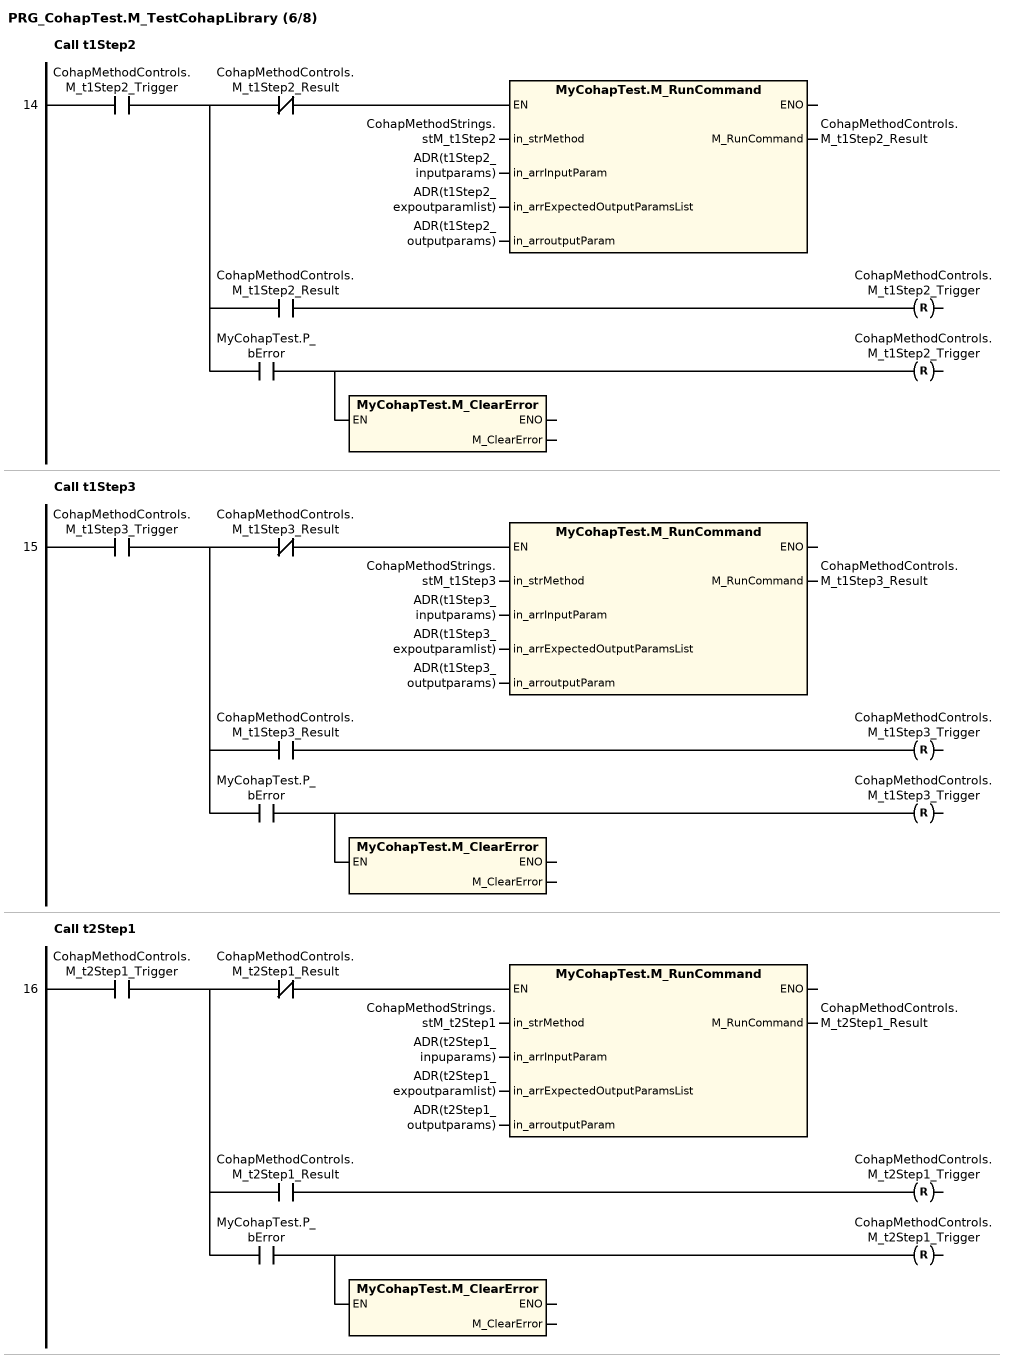
// NETWORK 14: Call t1Step2
_w27 := CohapMethodControls.M_t1Step2_Trigger;
IF _w27 AND NOT CohapMethodControls.M_t1Step2_Result THEN
    CohapMethodControls.M_t1Step2_Result := MyCohapTest.M_RunCommand(in_strMethod := CohapMethodStrings.stM_t1Step2, in_arrInputParam := ADR(t1Step2_inputparams), in_arrExpectedOutputParamsList := ADR(t1Step2_expoutparamlist), in_arroutputParam := ADR(t1Step2_outputparams));
END_IF
CohapMethodControls.M_t1Step2_Trigger R= _w27 AND CohapMethodControls.M_t1Step2_Result;
_w28 := _w27 AND MyCohapTest.P_bError;
CohapMethodControls.M_t1Step2_Trigger R= _w28;
IF _w28 THEN MyCohapTest.M_ClearError(); END_IF

// NETWORK 15: Call t1Step3
_w29 := CohapMethodControls.M_t1Step3_Trigger;
IF _w29 AND NOT CohapMethodControls.M_t1Step3_Result THEN
    CohapMethodControls.M_t1Step3_Result := MyCohapTest.M_RunCommand(in_strMethod := CohapMethodStrings.stM_t1Step3, in_arrInputParam := ADR(t1Step3_inputparams), in_arrExpectedOutputParamsList := ADR(t1Step3_expoutparamlist), in_arroutputParam := ADR(t1Step3_outputparams));
END_IF
CohapMethodControls.M_t1Step3_Trigger R= _w29 AND CohapMethodControls.M_t1Step3_Result;
_w30 := _w29 AND MyCohapTest.P_bError;
CohapMethodControls.M_t1Step3_Trigger R= _w30;
IF _w30 THEN MyCohapTest.M_ClearError(); END_IF

// NETWORK 16: Call t2Step1
_w31 := CohapMethodControls.M_t2Step1_Trigger;
IF _w31 AND NOT CohapMethodControls.M_t2Step1_Result THEN
    CohapMethodControls.M_t2Step1_Result := MyCohapTest.M_RunCommand(in_strMethod := CohapMethodStrings.stM_t2Step1, in_arrInputParam := ADR(t2Step1_inpuparams), in_arrExpectedOutputParamsList := ADR(t2Step1_expoutparamlist), in_arroutputParam := ADR(t2Step1_outputparams));
END_IF
CohapMethodControls.M_t2Step1_Trigger R= _w31 AND CohapMethodControls.M_t2Step1_Result;
_w32 := _w31 AND MyCohapTest.P_bError;
CohapMethodControls.M_t2Step1_Trigger R= _w32;
IF _w32 THEN MyCohapTest.M_ClearError(); END_IF

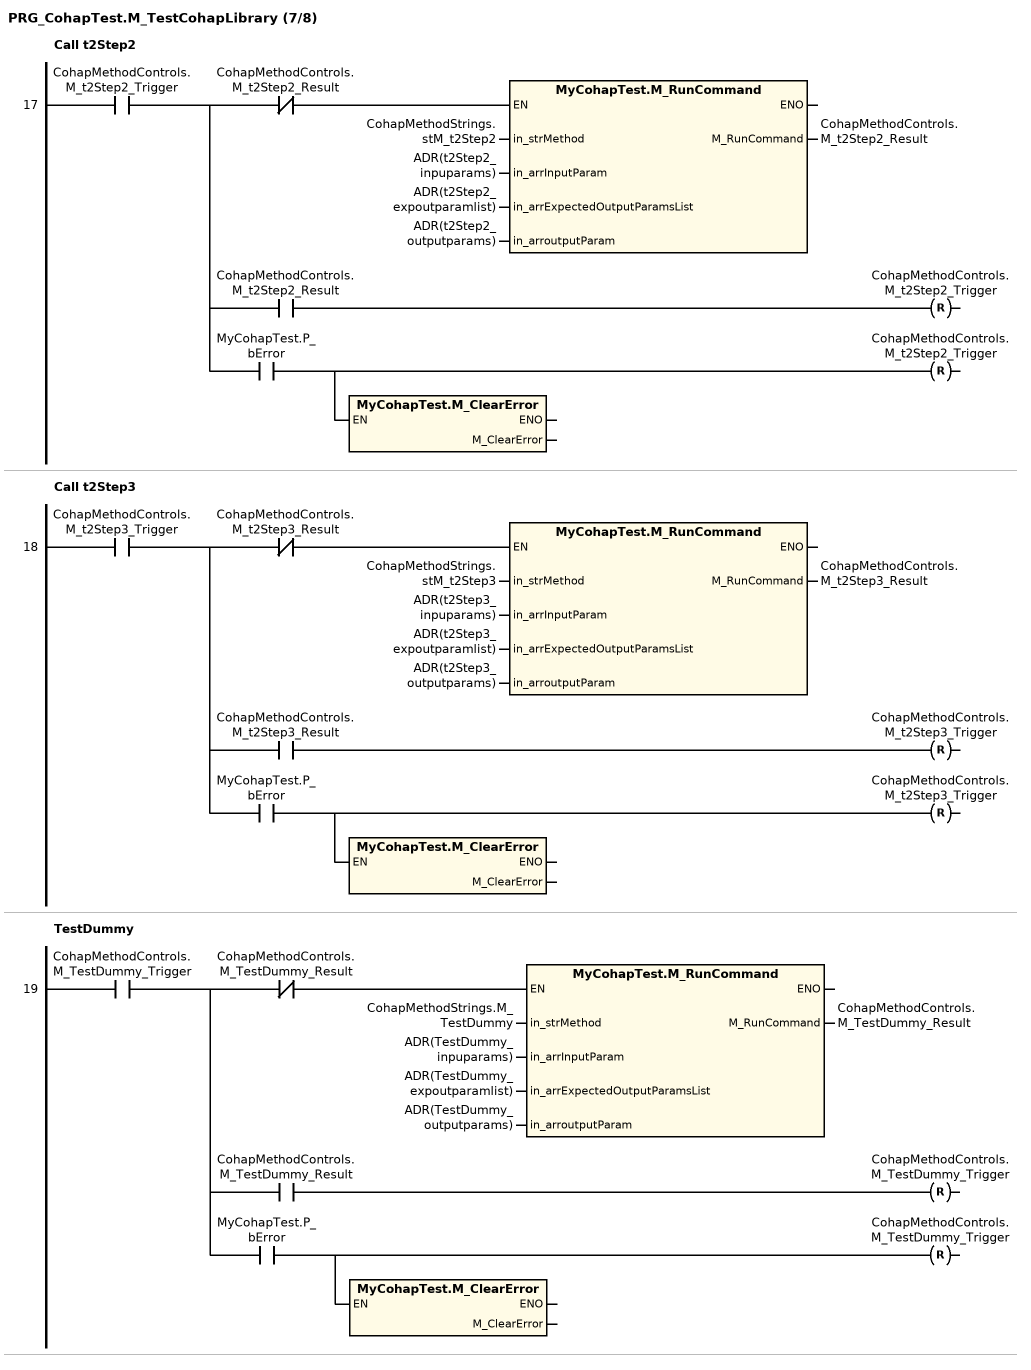
// NETWORK 17: Call t2Step2
_w33 := CohapMethodControls.M_t2Step2_Trigger;
IF _w33 AND NOT CohapMethodControls.M_t2Step2_Result THEN
    CohapMethodControls.M_t2Step2_Result := MyCohapTest.M_RunCommand(in_strMethod := CohapMethodStrings.stM_t2Step2, in_arrInputParam := ADR(t2Step2_inpuparams), in_arrExpectedOutputParamsList := ADR(t2Step2_expoutparamlist), in_arroutputParam := ADR(t2Step2_outputparams));
END_IF
CohapMethodControls.M_t2Step2_Trigger R= _w33 AND CohapMethodControls.M_t2Step2_Result;
_w34 := _w33 AND MyCohapTest.P_bError;
CohapMethodControls.M_t2Step2_Trigger R= _w34;
IF _w34 THEN MyCohapTest.M_ClearError(); END_IF

// NETWORK 18: Call t2Step3
_w35 := CohapMethodControls.M_t2Step3_Trigger;
IF _w35 AND NOT CohapMethodControls.M_t2Step3_Result THEN
    CohapMethodControls.M_t2Step3_Result := MyCohapTest.M_RunCommand(in_strMethod := CohapMethodStrings.stM_t2Step3, in_arrInputParam := ADR(t2Step3_inpuparams), in_arrExpectedOutputParamsList := ADR(t2Step3_expoutparamlist), in_arroutputParam := ADR(t2Step3_outputparams));
END_IF
CohapMethodControls.M_t2Step3_Trigger R= _w35 AND CohapMethodControls.M_t2Step3_Result;
_w36 := _w35 AND MyCohapTest.P_bError;
CohapMethodControls.M_t2Step3_Trigger R= _w36;
IF _w36 THEN MyCohapTest.M_ClearError(); END_IF

// NETWORK 19: TestDummy
_w37 := CohapMethodControls.M_TestDummy_Trigger;
IF _w37 AND NOT CohapMethodControls.M_TestDummy_Result THEN
    CohapMethodControls.M_TestDummy_Result := MyCohapTest.M_RunCommand(in_strMethod := CohapMethodStrings.M_TestDummy, in_arrInputParam := ADR(TestDummy_inpuparams), in_arrExpectedOutputParamsList := ADR(TestDummy_expoutparamlist), in_arroutputParam := ADR(TestDummy_outputparams));
END_IF
CohapMethodControls.M_TestDummy_Trigger R= _w37 AND CohapMethodControls.M_TestDummy_Result;
_w38 := _w37 AND MyCohapTest.P_bError;
CohapMethodControls.M_TestDummy_Trigger R= _w38;
IF _w38 THEN MyCohapTest.M_ClearError(); END_IF

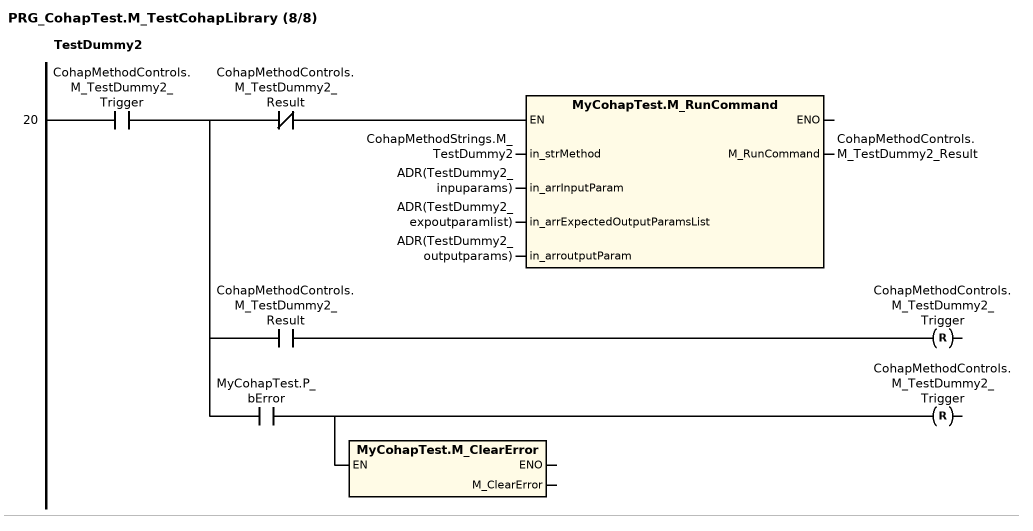
// NETWORK 20: TestDummy2
_w39 := CohapMethodControls.M_TestDummy2_Trigger;
IF _w39 AND NOT CohapMethodControls.M_TestDummy2_Result THEN
    CohapMethodControls.M_TestDummy2_Result := MyCohapTest.M_RunCommand(in_strMethod := CohapMethodStrings.M_TestDummy2, in_arrInputParam := ADR(TestDummy2_inpuparams), in_arrExpectedOutputParamsList := ADR(TestDummy2_expoutparamlist), in_arroutputParam := ADR(TestDummy2_outputparams));
END_IF
CohapMethodControls.M_TestDummy2_Trigger R= _w39 AND CohapMethodControls.M_TestDummy2_Result;
_w40 := _w39 AND MyCohapTest.P_bError;
CohapMethodControls.M_TestDummy2_Trigger R= _w40;
IF _w40 THEN MyCohapTest.M_ClearError(); END_IF
END_METHOD

END_PROGRAM

(* stored: Version 1.1.0.1, ProductVersion 3.1.4024.12
   POU PRG_CohapTest: Id {a44faab2-c81f-4a9e-9acb-c7e11c904ce6}, SpecialFunc None
   Action A_InitCohapMethodParams: Id {338b2860-1dc4-47ff-9b38-e01ddb531ef1}
   Method M_TestCohapLibrary: Id {03d0f1cf-5945-40d8-8fae-1fb0593baa2d} *)
